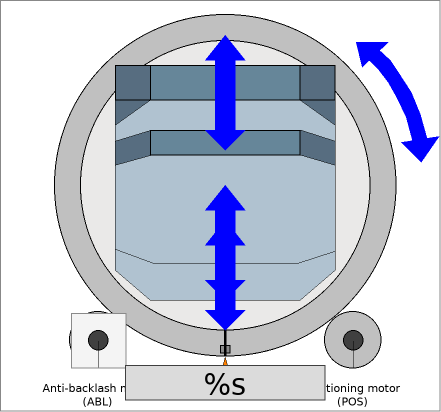
VISUALIZATION VISU_M3Figure  // 441x412
VAR_IN_OUT
    m3 : M3;
    widget : M3Widget;
    hideDetails : BOOL;
END_VAR
    Rectangle (220,365 10x23), invisible if: hideDetails
        p2858320360: widget.rotation.negativeLimitAngle
    Ellipse (54,14 342x342)
    Ellipse (80,40 290x290)
    Rectangle (155,175 140x30), "%s", text variable: m3.config.knownPositions.cassegrain.name, colour toggle: widget.cassegrainActive
    Polygon (150,100) (115,125) (115,100) (150,75) (300,75) (335,100) (335,125) (300,100), invisible if: widget.translation.hide_nasmyth
        p2858320360: widget.rotation.mirrorAngle
    Polygon (150,300) (115,270) (115,125) (150,100) (300,100) (335,125) (335,270) (300,300), invisible if: widget.translation.hide_nasmyth
        p2858320360: widget.rotation.mirrorAngle
    Rectangle (150,75 150x25), invisible if: widget.translation.hide_nasmyth
        p2858320360: widget.rotation.mirrorAngle
    Ellipse (324,311 57x57), invisible if: hideDetails
    Ellipse (343,330 20x20), invisible if: hideDetails
    Polygon (353,341) (353,367) (353,367) (353,341), invisible if: hideDetails
        p2858320360: m3.parts.rotation.parts.positioningHallAxis.actPos.degrees.value
    Ellipse (69,311 57x57), invisible if: hideDetails
    Ellipse (220,375 10x10), colour toggle: m3.parts.rotation.negativeLimitSwitchActive, invisible if: hideDetails
        p2858320360: widget.rotation.negativeLimitAngle
    Rectangle (220,365 10x23), invisible if: hideDetails
        p2858320360: widget.rotation.positiveLimitAngle
    Ellipse (220,375 10x10), colour toggle: m3.parts.rotation.positiveLimitSwitchActive, invisible if: hideDetails
        p2858320360: widget.rotation.positiveLimitAngle
    Rectangle (220,345 10x8), invisible if: hideDetails
        p2858320360: widget.rotation.hardwareLimitAngle
    Polygon (226,330) (226,356) (224,356) (224,330)
        p2858320360: widget.rotation.mirrorAngle
    Polygon (225,357) (230,375) (220,375)
        p2858320360: widget.rotation.targetAngle
    Pie (71,313 55x55), invisible if: hideDetails
        p426801730: widget.rotation.offsetStartAngle
        p2124672552: widget.rotation.offsetEndAngle
        p2858320360: widget.rotation.offsetAngle
    Ellipse (88,330 20x20), invisible if: hideDetails
    Polygon (98,341) (98,367) (98,367) (98,341), invisible if: hideDetails
        p2858320360: m3.parts.rotation.parts.antiBacklashAxis.actPos.degrees.value
    Label (35,380 125x30), "Anti-backlash motor (ABL)", invisible if: hideDetails
    Label (290,380 125x30), "Positioning motor (POS)", invisible if: hideDetails
    Polygon (151,155) (115,165) (115,141) (151,130) (301,130) (335,141) (335,165) (301,155), invisible if: widget.translation.hide_half
        p2858320360: widget.rotation.mirrorAngle
    Rectangle (150,130 150x25), invisible if: widget.translation.hide_half
        p2858320360: widget.rotation.mirrorAngle
    Polygon (153,263) (115,249) (115,165) (151,155) (301,155) (335,165) (335,251) (298,263), invisible if: widget.translation.hide_half
        p2858320360: widget.rotation.mirrorAngle
    Rectangle (125,365 200x35), "%s", text variable: m3.config.knownPositions.nasmythA.name, colour toggle: widget.nasmythAActive
        p2858320360: widget.nasmythAAngle
    Rectangle (125,365 200x35), "%s", text variable: m3.config.knownPositions.nasmythB.name, colour toggle: widget.nasmythBActive
        p2858320360: widget.nasmythBAngle
    Polygon (439,136) (421,162) (401,142), invisible if: NOT m3.parts.rotation.parts.positioningAxis.statuses.motionStatus.backward
    Polygon (388,42) (362,67) (356,42), invisible if: NOT m3.parts.rotation.parts.positioningAxis.statuses.motionStatus.forward
    Polygon (367,58) (377,48) (390,60) (398,72) (411,92) (420,114) (427,139) (413,143) (406,117) (397,98) (388,82) (378,69), invisible if: m3.parts.rotation.parts.positioningAxis.statuses.motionStatus.standstill
    Polygon (245,245) (225,220) (205,245) (215,245) (215,290) (235,290) (235,245), invisible if: widget.translation.hide_nasmyth_decreasing
        p2858320360: widget.rotation.mirrorAngle
    Polygon (245,310) (225,330) (205,310) (215,310) (215,280) (235,280) (235,310), invisible if: widget.translation.hide_nasmyth_increasing
        p2858320360: widget.rotation.mirrorAngle
    Polygon (245,280) (225,300) (205,280) (215,280) (215,250) (235,250) (235,280), invisible if: widget.translation.hide_half_increasing
        p2858320360: widget.rotation.mirrorAngle
    Polygon (245,210) (225,185) (205,210) (215,210) (215,255) (235,255) (235,210), invisible if: widget.translation.hide_half_decreasing
        p2858320360: widget.rotation.mirrorAngle
    Rectangle (115,65 220x35), invisible if: widget.translation.hide_cassegrain
        p2858320360: widget.rotation.mirrorAngle
    Rectangle (150,65 150x35), invisible if: widget.translation.hide_cassegrain
        p2858320360: widget.rotation.mirrorAngle
    Polygon (245,60) (225,35) (205,60) (215,60) (215,100) (235,100) (235,60), invisible if: widget.translation.hide_cassegrain_decreasing
        p2858320360: widget.rotation.mirrorAngle
    Polygon (245,130) (225,150) (205,130) (215,130) (215,100) (235,100) (235,130), invisible if: widget.translation.hide_cassegrain_increasing
        p2858320360: widget.rotation.mirrorAngle
END_VISUALIZATION

(* stored: Version 1.1.0.1, ProductVersion 3.1.4018.2
   Visu VISU_M3Figure: Id {a3ef0b9d-3f9c-4fc0-8dc3-544c8cd1d4aa} *)
